Staubli VAL3: Variables.pgx

program Variables()
begin
  jInit = {0,0,0,0,0,0}
  jDest = {0,90,-90,0,0,0}
  pCarre1 = {{0,600,500,0,0,0}, {sfree, efree, wfree}}
  pCarre2 = {{-500,0,500,0,0,0}, {sfree, efree, wfree}}
  pCarre3 = {{0,-500,500,0,0,0}, {sfree, efree, wfree}}
  pCarre4 = {{500,0,500,0,0,0}, {sfree, efree, wfree}}
end
